(* CoDeSys 2.3.9.31 project: mainProject.pro *)
(* Libraries: STANDARD.LIB 5.6.98 11:03:02 *)

(* Task configuration *)
TASK Standard (PRIORITY := 0, INTERVAL := T#10ms);
	MAIN
END_TASK

(* Global variable list: Global_Variables *)
VAR_GLOBAL

	(* Выключатели, датчики, освещение и клапаны по комнатам *)
	(* Щит 0 *)
	IN_CTL_BTN_1: BOOL; (* Выключатель основной *)

	(* Кухня 1 *)
	IN_KTN_BTN_1: BOOL; (* Выключатель основной *)
	IN_KTN_BTN_2: BOOL; (* Выключатель для вытяжки *)
	IN_KTN_DTR_1: BOOL; (* Датчик протечек *)

	OUT_KTN_LIGHT_1: BOOL; (* Свет основной *)
	OUT_KTN_LIGHT_2: BOOL; (* Свет второстепенный (подсветка) *)
	OUT_KTN_FAN_1: BOOL; (* Вытяжка *)

	(* Балкон 2 *)
	IN_BLKN_BTN_1: BOOL; (* Выключатель *)
	OUT_BLKN_LIGHT_1: BOOL; (* Свет *)

	(* Гостиная 3 *)
	IN_LVG_BTN_1: BOOL; (* Выключатель *)
	IN_LVG_BTN_2: BOOL; (* Выключатель на рабочем месте *)
	OUT_LVG_LIGHT_1: BOOL; (* Свет основной *)
	OUT_LVG_LIGHT_2: BOOL; (* Свет второстепенный *)

	(* Спальная 4 *)
	IN_BDR_BTN_1: BOOL; (* Выключатель *)
	IN_BDR_BTN_2: BOOL; (* Выключатель над кроватью *)
	IN_BDR_BTN_3: BOOL; (* Выключатель над кроватью *)
	OUT_BDR_LIGHT_1: BOOL; (* Свет *)
	OUT_BDR_LIGHT_2: BOOL; (* Свет второстепенный *)
	OUT_BDR_LIGHT_3: BOOL; (* Свет над кроватью (торшер) *)
	OUT_BDR_LIGHT_4: BOOL; (* Свет над кроватью (торшер) *)

	(* Ванная большая 5 *)
	IN_BMB_BTN_1: BOOL; (* Выключатель основной *)
	IN_BMB_BTN_2: BOOL; (* Выключатель около зеркала *)
	IN_BMB_DTR_1: BOOL; (* Датчик протечек *)
	OUT_BMB_LIGHT_1: BOOL; (* Свет основной *)
	OUT_BMB_LIGHT_2: BOOL; (* Свет около зеркала *)
	OUT_BMB_FAN_1: BOOL; (* Вытяжка *)
	OUT_BMB_VLV_1: BOOL; (* Вентиль *)
	OUT_BMB_VLV_2: BOOL; (* Вентиль *)

	(* Детская 6 *)
	IN_CHLD_BTN_1: BOOL; (* Выключатель *)
	OUT_CHLD_LIGHT_1: BOOL; (* Свет основной *)
	OUT_CHLD_LIGHT_2: BOOL; (* Свет второстепенный *)

	(* Коридор 7 *)
	IN_HLL_BTN_1: BOOL; (* Проходной выключатель *)
	IN_HLL_BTN_2: BOOL; (* Проходной выключатель *)
	IN_HLL_BTN_3: BOOL; (* Выключатель на зеркало *)
	OUT_HLL_LIGHT_1: BOOL; (* Свет основной *)
	OUT_HLL_LIGHT_2: BOOL; (* Свет второстепенный *)
	OUT_HLL_LIGHT_3: BOOL; (* Свет зеркало *)

	(* Ванная малая 8 *)
	IN_BMS_BTN_1: BOOL; (* Выключатель *)
	IN_BMS_DTR_1: BOOL; (* Датчик протечек *)
	OUT_BMS_LIGHT_1: BOOL; (* Свет *)
	OUT_BMS_FAN_1: BOOL; (* Вытяжка *)
	OUT_BMS_VLV_1: BOOL; (* Вентиль *)
	OUT_BMS_VLV_2: BOOL; (* Вентиль *)

	(* Розетки *)
	(* Щит *)
	G_OUT_0_SOCKET_G2: BOOL; (* Неотключаемые (рядом со щитком, роутер, сервер и т.п.) *)

	(* Кухня и балкон *)
	G_OUT_1_2_SOCKET_G1: BOOL; (* Общие *)
	G_OUT_1_2_SOCKET_G2: BOOL; (* Неотключаемые (холодильник)*)
	G_OUT_1_2_SOCKET_G3: BOOL; (* Посудомойка *)
	G_OUT_1_2_SOCKET_G4: BOOL; (* Плита, 380В *)

	(* Гостиная и спальня *)
	G_OUT_3_4_SOCKET_G1: BOOL; (* Общие *)
	G_OUT_3_4_SOCKET_G2: BOOL; (* Неотключаемые (компьютер) *)

	(* Ванная большая *)
	G_OUT_5_SOCKET_G1: BOOL; (* Общие *)
	G_OUT_5_SOCKET_G2: BOOL; (* Стиральная машина *)
	G_OUT_5_SOCKET_G3: BOOL; (* Резерв на бойлер и (или) баню *)

	(* Коридор и детская *)
	G_OUT_6_7_SOCKET_G1: BOOL; (* Общие *)

END_VAR

(* Global variable list: TwinCAT_Import *)
VAR_GLOBAL (* DO NOT CHANGE THIS SHEET MANUALLY! *)
	PlcInVar_0	AT %QB128:	USINT;
	PlcInVar_1	AT %QB129:	USINT;
	PlcInVar_2	AT %QB130:	USINT;
	PlcInVar_3	AT %QB131:	USINT;
	PlcInVar_4	AT %QB132:	USINT;
	PlcInVar_5	AT %QB133:	USINT;
	PlcInVar_6	AT %QB134:	USINT;
	PlcInVar_7	AT %QB135:	USINT;
	PlcInVar_8	AT %QB136:	USINT;
	PlcInVar_9	AT %QB137:	USINT;
	PlcInVar_10	AT %QB138:	USINT;
	PlcInVar_11	AT %QB139:	USINT;
	PlcInVar_12	AT %QB140:	USINT;
	PlcInVar_13	AT %QB141:	USINT;
	PlcInVar_14	AT %QB142:	USINT;
	PlcInVar_15	AT %QB143:	USINT;
	PlcOutVar_0	AT %IB128:	USINT;
	PlcOutVar_1	AT %IB129:	USINT;
	PlcOutVar_2	AT %IB130:	USINT;
	PlcOutVar_3	AT %IB131:	USINT;
	PlcOutVar_4	AT %IB132:	USINT;
	PlcOutVar_5	AT %IB133:	USINT;
	PlcOutVar_6	AT %IB134:	USINT;
	PlcOutVar_7	AT %IB135:	USINT;
	PlcOutVar_8	AT %IB136:	USINT;
	PlcOutVar_9	AT %IB137:	USINT;
	PlcOutVar_10	AT %IB138:	USINT;
	PlcOutVar_11	AT %IB139:	USINT;
	PlcOutVar_12	AT %IB140:	USINT;
	PlcOutVar_13	AT %IB141:	USINT;
	PlcOutVar_14	AT %IB142:	USINT;
	PlcOutVar_15	AT %IB143:	USINT;
	Term_2_KL2408_1_Output	AT %QX0.0:	BOOL;
	Term_2_KL2408_2_Output	AT %QX0.1:	BOOL;
	Term_2_KL2408_3_Output	AT %QX0.2:	BOOL;
	Term_2_KL2408_4_Output	AT %QX0.3:	BOOL;
	Term_2_KL2408_5_Output	AT %QX0.4:	BOOL;
	Term_2_KL2408_6_Output	AT %QX0.5:	BOOL;
	Term_2_KL2408_7_Output	AT %QX0.6:	BOOL;
	Term_2_KL2408_8_Output	AT %QX0.7:	BOOL;
	Term_3_KL2408_1_Output	AT %QX1.0:	BOOL;
	Term_3_KL2408_2_Output	AT %QX1.1:	BOOL;
	Term_3_KL2408_3_Output	AT %QX1.2:	BOOL;
	Term_3_KL2408_4_Output	AT %QX1.3:	BOOL;
	Term_3_KL2408_5_Output	AT %QX1.4:	BOOL;
	Term_3_KL2408_6_Output	AT %QX1.5:	BOOL;
	Term_3_KL2408_7_Output	AT %QX1.6:	BOOL;
	Term_3_KL2408_8_Output	AT %QX1.7:	BOOL;
	Term_4_KL2408_1_Output	AT %QX2.0:	BOOL;
	Term_4_KL2408_2_Output	AT %QX2.1:	BOOL;
	Term_4_KL2408_3_Output	AT %QX2.2:	BOOL;
	Term_4_KL2408_4_Output	AT %QX2.3:	BOOL;
	Term_4_KL2408_5_Output	AT %QX2.4:	BOOL;
	Term_4_KL2408_6_Output	AT %QX2.5:	BOOL;
	Term_4_KL2408_7_Output	AT %QX2.6:	BOOL;
	Term_4_KL2408_8_Output	AT %QX2.7:	BOOL;
	Term_5_KL2408_1_Output	AT %QX3.0:	BOOL;
	Term_5_KL2408_2_Output	AT %QX3.1:	BOOL;
	Term_5_KL2408_3_Output	AT %QX3.2:	BOOL;
	Term_5_KL2408_4_Output	AT %QX3.3:	BOOL;
	Term_5_KL2408_5_Output	AT %QX3.4:	BOOL;
	Term_5_KL2408_6_Output	AT %QX3.5:	BOOL;
	Term_5_KL2408_7_Output	AT %QX3.6:	BOOL;
	Term_5_KL2408_8_Output	AT %QX3.7:	BOOL;
	Term_6_KL2408_1_Output	AT %QX4.0:	BOOL;
	Term_6_KL2408_2_Output	AT %QX4.1:	BOOL;
	Term_6_KL2408_3_Output	AT %QX4.2:	BOOL;
	Term_6_KL2408_4_Output	AT %QX4.3:	BOOL;
	Term_6_KL2408_5_Output	AT %QX4.4:	BOOL;
	Term_6_KL2408_6_Output	AT %QX4.5:	BOOL;
	Term_6_KL2408_7_Output	AT %QX4.6:	BOOL;
	Term_6_KL2408_8_Output	AT %QX4.7:	BOOL;
	Term_7_KL1408_1_Input	AT %IX0.0:	BOOL;
	Term_7_KL1408_2_Input	AT %IX0.1:	BOOL;
	Term_7_KL1408_3_Input	AT %IX0.2:	BOOL;
	Term_7_KL1408_4_Input	AT %IX0.3:	BOOL;
	Term_7_KL1408_5_Input	AT %IX0.4:	BOOL;
	Term_7_KL1408_6_Input	AT %IX0.5:	BOOL;
	Term_7_KL1408_7_Input	AT %IX0.6:	BOOL;
	Term_7_KL1408_8_Input	AT %IX0.7:	BOOL;
	Term_8_KL1408_1_Input	AT %IX1.0:	BOOL;
	Term_8_KL1408_2_Input	AT %IX1.1:	BOOL;
	Term_8_KL1408_3_Input	AT %IX1.2:	BOOL;
	Term_8_KL1408_4_Input	AT %IX1.3:	BOOL;
	Term_8_KL1408_5_Input	AT %IX1.4:	BOOL;
	Term_8_KL1408_6_Input	AT %IX1.5:	BOOL;
	Term_8_KL1408_7_Input	AT %IX1.6:	BOOL;
	Term_8_KL1408_8_Input	AT %IX1.7:	BOOL;
	Term_9_KL1408_1_Input	AT %IX2.0:	BOOL;
	Term_9_KL1408_2_Input	AT %IX2.1:	BOOL;
	Term_9_KL1408_3_Input	AT %IX2.2:	BOOL;
	Term_9_KL1408_4_Input	AT %IX2.3:	BOOL;
	Term_9_KL1408_5_Input	AT %IX2.4:	BOOL;
	Term_9_KL1408_6_Input	AT %IX2.5:	BOOL;
	Term_9_KL1408_7_Input	AT %IX2.6:	BOOL;
	Term_9_KL1408_8_Input	AT %IX2.7:	BOOL;
	Term_10_KL1408_1_Input	AT %IX3.0:	BOOL;
	Term_10_KL1408_2_Input	AT %IX3.1:	BOOL;
	Term_10_KL1408_3_Input	AT %IX3.2:	BOOL;
	Term_10_KL1408_4_Input	AT %IX3.3:	BOOL;
	Term_10_KL1408_5_Input	AT %IX3.4:	BOOL;
	Term_10_KL1408_6_Input	AT %IX3.5:	BOOL;
	Term_10_KL1408_7_Input	AT %IX3.6:	BOOL;
	Term_10_KL1408_8_Input	AT %IX3.7:	BOOL;
END_VAR

(* POU MAIN, ST *)
PROGRAM MAIN
VAR
	T_LONG_PRESS : TIME := t#1000ms;
END_VAR

END_PROGRAM
